      -Name "ICI_TYPE" -BusType "PIO" -VendorName "ABB"\
      -ProductName "IPS (ICI) unit"
#
EIO_UNIT:

      -Name "PIB" -UnitType "ICI_TYPE" -Bus "ICIBUS"\
      -UnitLabel "Process Interface Board" -PIO_Address "192.168.126.200"

      -Name "PibSaf" -UnitType "ICI_TYPE" -Bus "ICIBUS" -UnitLabel "Safety Unit"\
      -PIO_Address "192.168.126.200"

      -Name "SysComm" -UnitType "Virtual" -Bus "Virtual1"

      -Name "CommandIO" -UnitType "Virtual" -Bus "Virtual1"

      -Name "DummyIO" -UnitType "Virtual" -Bus "Virtual1"
#
EIO_SIGNAL:

      -Name "sdoAutoOn" -SignalType "DO" -Unit "SysComm" -UnitMap "0"

      -Name "sdoCycleOn" -SignalType "DO" -Unit "SysComm" -UnitMap "1"

      -Name "sdoEmStop" -SignalType "DO" -Unit "SysComm" -UnitMap "2"

      -Name "sdoError" -SignalType "DO" -Unit "SysComm" -UnitMap "3"

      -Name "sdoMotOnState" -SignalType "DO" -Unit "SysComm" -UnitMap "4"

      -Name "sdoRunchOk" -SignalType "DO" -Unit "SysComm" -UnitMap "5"

      -Name "sdoMotorOn" -SignalType "DO" -Unit "SysComm" -UnitMap "6"

      -Name "sdoMotorOff" -SignalType "DO" -Unit "SysComm" -UnitMap "7"

      -Name "sdoStart" -SignalType "DO" -Unit "SysComm" -UnitMap "8"

      -Name "sdoStop" -SignalType "DO" -Unit "SysComm" -UnitMap "9"

      -Name "sdoResetError" -SignalType "DO" -Unit "SysComm" -UnitMap "10"

      -Name "sdoSysReset" -SignalType "DO" -Unit "SysComm" -UnitMap "11"

      -Name "sdoStartMain" -SignalType "DO" -Unit "SysComm" -UnitMap "12"

      -Name "sdoManRedSpeed" -SignalType "DO" -Unit "SysComm" -UnitMap "13"

      -Name "sdoManFullSpeed" -SignalType "DO" -Unit "SysComm" -UnitMap "14"

      -Name "sdoSwitchInAuto" -SignalType "DO" -Unit "SysComm" -UnitMap "15"

      -Name "doPntRapidError" -SignalType "DO" -Unit "SysComm" -UnitMap "20"

      -Name "doAutoMode" -SignalType "DO" -Unit "SysComm" -UnitMap "21"

      -Name "doInitialized" -SignalType "DO" -Unit "SysComm" -UnitMap "22"

      -Name "doInModule" -SignalType "DO" -Unit "SysComm" -UnitMap "23" -Store

      -Name "doJobInProgress" -SignalType "DO" -Unit "SysComm" -UnitMap "24"\
      -Store

      -Name "doQueueNotEmpty" -SignalType "DO" -Unit "SysComm" -UnitMap "25"

      -Name "doQueueFull" -SignalType "DO" -Unit "SysComm" -UnitMap "26"

      -Name "doQueueExpedited" -SignalType "DO" -Unit "SysComm" -UnitMap "27"

      -Name "doQueuePause" -SignalType "DO" -Unit "SysComm" -UnitMap "28"

      -Name "doSpyStart" -SignalType "DO" -Unit "SysComm" -UnitMap "29"\
      -Access "ALL"

      -Name "doSpyStop" -SignalType "DO" -Unit "SysComm" -UnitMap "30"\
      -Access "ALL"

      -Name "doMtrlSupOn" -SignalType "DO" -Unit "SysComm" -UnitMap "31"

      -Name "doHomePos" -SignalType "DO" -Unit "SysComm" -UnitMap "32"\
      -Access "INTERNAL"

      -Name "doMtrlChangePos" -SignalType "DO" -Unit "SysComm" -UnitMap "33"\
      -Access "INTERNAL"

      -Name "doReadyPos" -SignalType "DO" -Unit "SysComm" -UnitMap "34"\
      -Access "INTERNAL"

      -Name "doUserPos" -SignalType "DO" -Unit "SysComm" -UnitMap "35"\
      -Access "INTERNAL"

      -Name "doModeChangeAck" -SignalType "DO" -Unit "SysComm" -UnitMap "36"

      -Name "doExStart" -SignalType "DO" -Unit "SysComm" -UnitMap "37"

      -Name "doCmdReady" -SignalType "DO" -Unit "SysComm" -UnitMap "38"

      -Name "doCmdExecuting" -SignalType "DO" -Unit "SysComm" -UnitMap "39"

      -Name "doTPUCmdReady" -SignalType "DO" -Unit "SysComm" -UnitMap "40"

      -Name "doGUICmdReady" -SignalType "DO" -Unit "SysComm" -UnitMap "41"

      -Name "doIntCommand" -SignalType "DO" -Unit "SysComm" -UnitMap "42"

      -Name "doDirectModule" -SignalType "DO" -Unit "SysComm" -UnitMap "43"

      -Name "doMainInMC" -SignalType "DO" -Unit "SysComm" -UnitMap "44"

      -Name "doPLCCmdReady" -SignalType "DO" -Unit "SysComm" -UnitMap "45"

      -Name "doRapidError" -SignalType "DO" -Unit "SysComm" -UnitMap "46"

      -Name "doStartVClock" -SignalType "DO" -Unit "SysComm" -UnitMap "47"\
      -Access "ALL"

      -Name "doUpdateVClock" -SignalType "DO" -Unit "SysComm" -UnitMap "48"\
      -Access "ALL"

      -Name "doPaintBackup" -SignalType "DO" -Unit "SysComm" -UnitMap "49"\
      -Access "ALL"

      -Name "AutomaticMode" -SignalType "DO" -Unit "DummyIO" -UnitMap "0"\
      -Access "RAPIDONLY"

      -Name "MasterGranted" -SignalType "DO" -Unit "DummyIO" -UnitMap "1"\
      -Access "RAPIDONLY"

      -Name "RunChainClosed" -SignalType "DO" -Unit "DummyIO" -UnitMap "2"\
      -Access "RAPIDONLY"

      -Name "RobotError" -SignalType "DO" -Unit "DummyIO" -UnitMap "3"\
      -Access "RAPIDONLY"

      -Name "JobInProgress" -SignalType "DO" -Unit "DummyIO" -UnitMap "4"\
      -Access "RAPIDONLY"

      -Name "JobPending" -SignalType "DO" -Unit "DummyIO" -UnitMap "5"\
      -Access "RAPIDONLY"

      -Name "ReadyHighPri" -SignalType "DO" -Unit "DummyIO" -UnitMap "6"\
      -Access "RAPIDONLY"

      -Name "SystemRunning" -SignalType "DO" -Unit "DummyIO" -UnitMap "7"\
      -Access "RAPIDONLY"

      -Name "MtrlChRunning" -SignalType "DO" -Unit "DummyIO" -UnitMap "8"\
      -Access "RAPIDONLY"

      -Name "MtrlChangeOn" -SignalType "DO" -Unit "DummyIO" -UnitMap "9"\
      -Access "RAPIDONLY"

      -Name "MtrlSupplyEna" -SignalType "DO" -Unit "DummyIO" -UnitMap "10"\
      -Access "RAPIDONLY"

      -Name "MtrlSupplyError" -SignalType "DO" -Unit "DummyIO" -UnitMap "11"\
      -Access "RAPIDONLY"

      -Name "AppEnabled" -SignalType "DO" -Unit "DummyIO" -UnitMap "12"\
      -Access "RAPIDONLY"

      -Name "AppError" -SignalType "DO" -Unit "DummyIO" -UnitMap "13"\
      -Access "RAPIDONLY"

      -Name "HVEnabled" -SignalType "DO" -Unit "DummyIO" -UnitMap "14"\
      -Access "RAPIDONLY"

      -Name "HVError" -SignalType "DO" -Unit "DummyIO" -UnitMap "15"\
      -Access "RAPIDONLY"

      -Name "HeartBeat" -SignalType "DO" -Unit "DummyIO" -UnitMap "16"\
      -Access "RAPIDONLY"

      -Name "ConveyorHoldReq" -SignalType "DO" -Unit "DummyIO" -UnitMap "17"\
      -Access "RAPIDONLY"

      -Name "PotLifeTimeOut" -SignalType "DO" -Unit "DummyIO" -UnitMap "18"\
      -Access "RAPIDONLY"

      -Name "HomePos" -SignalType "DO" -Unit "DummyIO" -UnitMap "19"\
      -Access "RAPIDONLY"

      -Name "MtrlChangePos" -SignalType "DO" -Unit "DummyIO" -UnitMap "20"\
      -Access "RAPIDONLY"

      -Name "ReadyPos" -SignalType "DO" -Unit "DummyIO" -UnitMap "21"\
      -Access "RAPIDONLY"

      -Name "UserPos" -SignalType "DO" -Unit "DummyIO" -UnitMap "22"\
      -Access "RAPIDONLY"

      -Name "ReposFinished" -SignalType "DO" -Unit "DummyIO" -UnitMap "23"\
      -Access "RAPIDONLY"

      -Name "EmergencyStop" -SignalType "DO" -Unit "DummyIO" -UnitMap "24"\
      -Access "RAPIDONLY"

      -Name "JobComplete" -SignalType "DO" -Unit "DummyIO" -UnitMap "25"\
      -Access "RAPIDONLY"

      -Name "ManualMode" -SignalType "DO" -Unit "DummyIO" -UnitMap "26"\
      -Access "RAPIDONLY"

      -Name "ReadyToReceive" -SignalType "DO" -Unit "DummyIO" -UnitMap "27"\
      -Access "RAPIDONLY"

      -Name "MotorOn" -SignalType "DO" -Unit "DummyIO" -UnitMap "28"\
      -Access "RAPIDONLY"

      -Name "ProgramAck" -SignalType "DO" -Unit "DummyIO" -UnitMap "30"\
      -Access "RAPIDONLY"

      -Name "ProgramLoaded" -SignalType "DO" -Unit "DummyIO" -UnitMap "31"\
      -Access "RAPIDONLY"

      -Name "InModule" -SignalType "DO" -Unit "DummyIO" -UnitMap "69"\
      -Access "RAPIDONLY"

      -Name "ObjConnected" -SignalType "DO" -Unit "DummyIO" -UnitMap "70"\
      -Access "RAPIDONLY"

      -Name "ConveyorRunning" -SignalType "DO" -Unit "DummyIO" -UnitMap "71"\
      -Access "RAPIDONLY"

      -Name "CBSMotorOn" -SignalType "DO" -Unit "DummyIO" -UnitMap "72"\
      -Access "RAPIDONLY"

      -Name "PotLifeWarning" -SignalType "DO" -Unit "DummyIO" -UnitMap "73"\
      -Access "RAPIDONLY"

      -Name "GoingToAuto" -SignalType "DO" -Unit "DummyIO" -UnitMap "74"\
      -Access "RAPIDONLY"

      -Name "diModeChangeAck" -SignalType "DI" -Unit "SysComm" -UnitMap "1"

      -Name "A1Enable" -SignalType "DO" -Unit "SysComm" -UnitMap "100"\
      -Access "ALL"

      -Name "A1Error" -SignalType "DO" -Unit "SysComm" -UnitMap "101"\
      -Access "ALL"

      -Name "A1Material" -SignalType "GO" -Unit "SysComm" -UnitMap "110-119"\
      -Access "ALL"

      -Name "A1Brush" -SignalType "GO" -Unit "SysComm" -UnitMap "120-129"\
      -Access "ALL"

      -Name "A1BrushTabNdx" -SignalType "GO" -Unit "SysComm" -UnitMap "130-139"\
      -Access "ALL"

      -Name "A1Fluid" -SignalType "AO" -Unit "SysComm" -UnitMap "140-149"\
      -Access "ALL"

      -Name "A1HVErrNo" -SignalType "GO" -Unit "SysComm" -UnitMap "150-151"\
      -Access "ALL"

      -Name "A1HVEn" -SignalType "DO" -Unit "SysComm" -UnitMap "155"\
      -Access "ALL"

      -Name "SW_MOTOR_ON" -SignalType "DO" -Unit "PibSaf"\
      -UnitMap "Safety/OutPort1:SW_MOTOR_ON" -Access "INTERNAL"

      -Name "ReadyForMotorOn" -SignalType "DI" -Unit "PibSaf"\
      -UnitMap "Safety/InPort8:ReadyForMotorOn"

      -Name "MotorIsOn" -SignalType "DI" -Unit "PibSaf"\
      -UnitMap "Safety/InPort8:MotorIsOn"
#
EIO_CROSS:

      -Res "diModeChangeAck" -Act1 "doModeChangeAck"

      -Res "sdoManRedSpeed" -Act1 "MAN1" -Oper1 "AND" -Act2 "MAN2"

      -Res "sdoManFullSpeed" -Act1 "MANFS1" -Oper1 "AND" -Act2 "MANFS2"

      -Res "sdoSwitchInAuto" -Act1 "AUTO1" -Oper1 "AND" -Act2 "AUTO2"

      -Res "doAutoMode" -Act1 "sdoAutoOn" -Oper1 "AND" -Act2 "doInitialized"

      -Res "RobotError" -Act1 "sdoError" -Oper1 "OR" -Act2 "doPntRapidError"

      -Res "ReadyHighPri" -Act1 "sdoCycleOn" -Oper1 "AND"\
      -Act2 "doJobInProgress" -Act2_invert

      -Res "SystemRunning" -Act1 "sdoCycleOn" -Oper1 "AND" -Act2 "doQueuePause"\
      -Act2_invert

      -Res "doCmdReady" -Act1 "doPLCCmdReady" -Oper1 "OR" -Act2 "doTPUCmdReady"\
      -Oper2 "OR" -Act3 "doGUICmdReady" -Oper3 "OR" -Act4 "doIntCommand"

      -Res "AutomaticMode" -Act1 "doAutoMode"

      -Res "JobInProgress" -Act1 "doJobInProgress"

      -Res "JobPending" -Act1 "doQueueNotEmpty"

      -Res "EmergencyStop" -Act1 "sdoEmStop"

      -Res "MtrlSupplyEna" -Act1 "doMtrlSupOn"

      -Res "HomePos" -Act1 "doHomePos"

      -Res "MtrlChangePos" -Act1 "doMtrlChangePos"

      -Res "ReadyPos" -Act1 "doReadyPos"

      -Res "UserPos" -Act1 "doUserPos"

      -Res "AppEnabled" -Act1 "A1Enable"

      -Res "AppError" -Act1 "A1Error"

      -Res "A1HVEn" -Act1 "HVEnabled"

      -Res "InModule" -Act1 "doInModule"

      -Res "ManualMode" -Act1 "sdoManRedSpeed" -Oper1 "OR"\
      -Act2 "sdoManFullSpeed"

      -Res "ReadyToReceive" -Act1 "doInitialized" -Oper1 "AND"\
      -Act2 "doQueueFull" -Act2_invert

      -Res "GoingToAuto" -Act1 "sdoSwitchInAuto" -Oper1 "AND" -Act2 "sdoAutoOn"\
      -Act2_invert

      -Res "SW_MOTOR_ON" -Act1 "sdoMotorOn"

      -Res "RunChainClosed" -Act1 "ReadyForMotorOn"

      -Res "MotorOn" -Act1 "MotorIsOn"
#
EIO_ACCESS:

      -Name "All" -Rapid  -LocalManual  -LocalAuto  -RemoteManual  -RemoteAuto

      -Name "RAPIDONLY" -Rapid
#
SYSSIG_OUT:

      -Status "AutoOn" -Signal "sdoAutoOn"

      -Status "CycleOn" -Signal "sdoCycleOn"

      -Status "EmStop" -Signal "sdoEmStop"

      -Status "Error" -Signal "sdoError"

      -Status "MotOnState" -Signal "sdoMotOnState"

      -Status "RunchOk" -Signal "sdoRunchOk"
#
SYSSIG_IN:

      -Signal "sdoMotorOn" -Action "MotorOn"

      -Signal "sdoMotorOff" -Action "MotorOff"

      -Signal "sdoStart" -Action "Start"

      -Signal "sdoStop" -Action "Stop"

      -Signal "sdoResetError" -Action "ResetError"

      -Signal "sdoSysReset" -Action "SysReset"

      -Signal "sdoStartMain" -Action "StartMain"

      -Signal "doModeChangeAck" -Action "AckAutoMode"

--- Backups/Robo_open_v2/SYSPAR/PROC.cfg ---
PROC:CFG_1.0:5:0::
#
PW_SYSTEM:

      -name "PW_SYS" -pw_function "PW_FUNC"
#
PW_FUNCTION:

      -name "PW_FUNC" -do_repos_finished "ReposFinished"
